// TIA Portal V20 export
TYPE "typeCmInterfaceSoftCamVisionController"
// stored: Access Published, Namespace Unit1.Em6
   STRUCT
      homePos { ExternalWritable := 'False'} : "LER_typeSoftCamPosition";
      visionPos { ExternalWritable := 'False'} : "LER_typeSoftCamPosition";
      posistion2 { ExternalWritable := 'False'} : "LER_typeSoftCamPosition";
      posistion3 { ExternalWritable := 'False'} : "LER_typeSoftCamPosition";
      posistion4 { ExternalWritable := 'False'} : "LER_typeSoftCamPosition";
      posistion5 { ExternalWritable := 'False'} : "LER_typeSoftCamPosition";
      posistion6 { ExternalWritable := 'False'} : "LER_typeSoftCamPosition";
      posistion7 { ExternalWritable := 'False'} : "LER_typeSoftCamPosition";
      posistion8 { ExternalWritable := 'False'} : "LER_typeSoftCamPosition";
      posistion9 { ExternalWritable := 'False'} : "LER_typeSoftCamPosition";
      posistion10 { ExternalWritable := 'False'} : "LER_typeSoftCamPosition";
      posistion11 { ExternalWritable := 'False'} : "LER_typeSoftCamPosition";
      posistion12 { ExternalWritable := 'False'} : "LER_typeSoftCamPosition";
      posistion13 { ExternalWritable := 'False'} : "LER_typeSoftCamPosition";
      posistion14 { ExternalWritable := 'False'} : "LER_typeSoftCamPosition";
      posistion15 { ExternalWritable := 'False'} : "LER_typeSoftCamPosition";
   END_STRUCT;
END_TYPE
